// TIA Portal project "May dong chai_PLC_TiaPortal" (V16)
// Vorlageprojekt für das Buch mit Zielsystem S7-1200

(* hardware
DEVICE "S7-1200-Station_1"  S7-1200 Station
   slot 0: "Baugruppenträger_0"  Rack  V1.0
   slot 1: "PLC_1"  CPU 1211C DC/DC/DC  6ES7 211-1AE40-0XB0  V4.1
*)

// ===== PLC "PLC_1"  CPU 1211C DC/DC/DC =====

VAR_GLOBAL   // PLC tag table "Standard-Variablentabelle"
   "box-conveyor" AT %A0.0 : Bool;
   "start" AT %E0.0 : Bool;
   "stop" AT %E0.1 : Bool;
   "latch-relay" AT %M1.5 : Bool;
   "running" AT %M1.4 : Bool;
   "box-sensor" AT %I0.2 : Bool;
   "stop-state" AT %M1.6 : Bool;
   "can-conveyor" AT %Q0.1 : Bool;
   "can-sensor" AT %I0.3 : Bool;
   "Tag_10" AT %M2.0 : Bool;
   "1s" AT %M0.5 : Bool;
   "stop-light" AT %Q0.2 : Bool;
   "Clock_Byte" AT %MB0 : Byte;
   "Clock_10Hz" AT %M0.0 : Bool;
   "Clock_5Hz" AT %M0.1 : Bool;
   "Clock_2.5Hz" AT %M0.2 : Bool;
   "Clock_2Hz" AT %M0.3 : Bool;
   "Clock_1.25Hz" AT %M0.4 : Bool;
   "Clock_1Hz" AT %M0.5 : Bool;
   "Clock_0.625Hz" AT %M0.6 : Bool;
   "Clock_0.5Hz" AT %M0.7 : Bool;
END_VAR

// folder: System blocks/Program resources

DATA_BLOCK "counter1"   // DB1
{ S7_Optimized_Access := 'TRUE' }
AUTHOR : Simatic
FAMILY : IEC
NAME : CNTR
VERSION : 1.0
// stored: InstanceOfName IEC_COUNTER
"IEC_COUNTER"
BEGIN
END_DATA_BLOCK

DATA_BLOCK "counter2"   // DB2
{ S7_Optimized_Access := 'TRUE' }
AUTHOR : Simatic
FAMILY : IEC
NAME : CNTR
VERSION : 1.0
// stored: InstanceOfName IEC_COUNTER
"IEC_COUNTER"
BEGIN
END_DATA_BLOCK

DATA_BLOCK "timer1"   // DB3
{ S7_Optimized_Access := 'TRUE' }
AUTHOR : Simatic
FAMILY : IEC
NAME : IEC_TMR
VERSION : 1.0
// stored: InstanceOfName IEC_TIMER
"IEC_TIMER"
BEGIN
END_DATA_BLOCK

// folder: (top level)

FUNCTION "MHJ-PLC-Lab-Function-S71200" : Void   // FC9000, SCL
{ S7_Optimized_Access := 'TRUE' }
VERSION : 0.1
   VAR_TEMP
      rdTimeReturn : Int;
      outputTime : DTL;
      SyncVal : Byte;
      forVal : Int;
      forVal_2 : Int;
      Value : Byte;
   END_VAR
   VAR CONSTANT
      CompVal : Byte := 16#34;
      Value_01 : Byte := 16#11;
      Value_01_DW : DWord := 16#A165_D992;
      Value_02_DW : DWord := 16#58BE_4401;
   END_VAR
BEGIN

   #Value:=PEEK(area := 16#82,
        dbNumber := 0,
        byteOffset := 511);
   #Value := #Value + 1;

   POKE(area := 16#82,
        dbNumber := 0,
        byteOffset := 511,
        value := #Value);

   POKE(area:=16#81,
        dbNumber:=0,
        byteOffset:=1016,
        value:=#Value_01_DW);
   POKE(area := 16#81,
        dbNumber := 0,
        byteOffset := 1020,
        value := #Value_02_DW);

   POKE(area := 16#81,
        dbNumber := 0,
        byteOffset := 511,
        value := B#16#00);

   FOR #forVal := 0 TO 120 DO
       FOR #forVal_2:=0 TO 10 DO
           #rdTimeReturn:=RD_SYS_T(#outputTime);
           #rdTimeReturn := WR_SYS_T(#outputTime);
           #rdTimeReturn := RD_SYS_T(#outputTime);
           #rdTimeReturn := WR_SYS_T(#outputTime);
       END_FOR;
       #SyncVal:= PEEK(area := 16#81,
                      dbNumber := 0,
                      byteOffset := 511);
       IF #SyncVal = #CompVal THEN
          GOTO M_1;
       END_IF;
   END_FOR;
   RETURN;

   M_1:
   POKE(area := 16#81,
        dbNumber := 0,
        byteOffset := 511,
        value := B#16#0);
END_FUNCTION

ORGANIZATION_BLOCK "Main"   // OB1, LAD, ProgramCycle
TITLE = "Main Program Sweep (Cycle)"
{ S7_Optimized_Access := 'TRUE' }
VERSION : 0.1
   VAR_INPUT
      Initial_Call : Bool;   // Initial call of this OB
      Remanence : Bool;   // =True, if remanent data are available
   END_VAR
   VAR_TEMP   // added for the SCL form of the ladder/FBD networks
      _w1 : Bool;
      _w2 : Bool;
   END_VAR
BEGIN

REGION Network 1: Konnektierungsbaustein für PLC-Lab
   // Im Netzwerk 1 wird der Konnektierungsbaustein für PLC-Lab aufgerufen.
   // Dieser Aufruf darf nicht entfernt werden!
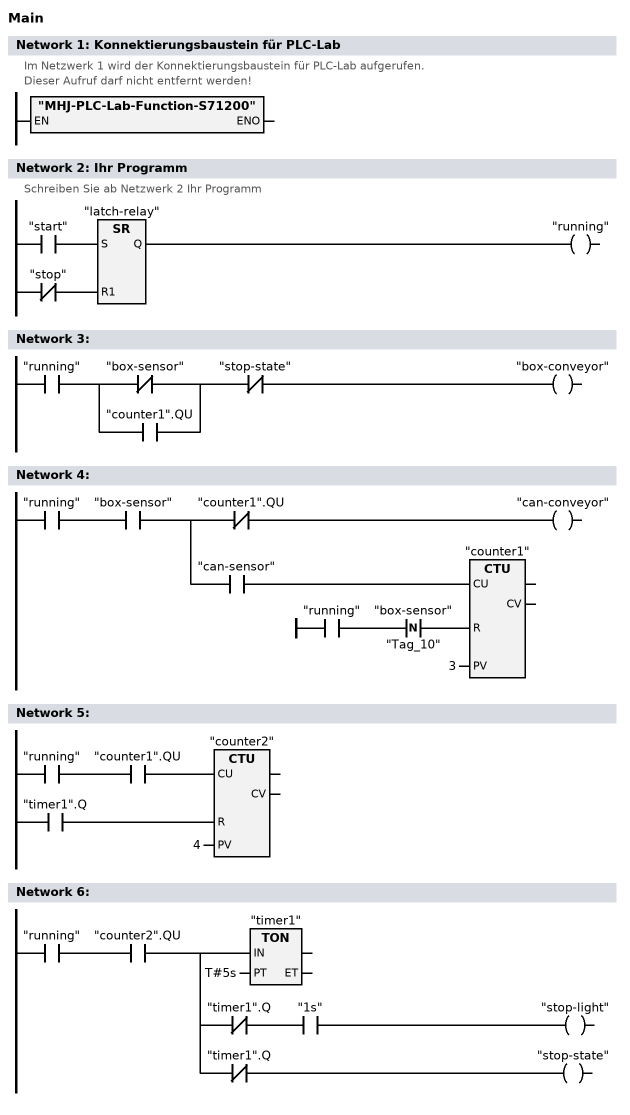
   RUNG wire#powerrail
      "MHJ-PLC-Lab-Function-S71200"()
   END_RUNG
   // the same network as SCL:
   "MHJ-PLC-Lab-Function-S71200"();
END_REGION

REGION Network 2: Ihr Programm
   // Schreiben Sie ab Netzwerk 2 Ihr Programm
   RUNG wire#powerrail
      Contact( "start" )
      S_SR(operand := "latch-relay", r1 := wire#w1)
      Coil( "running" )
   END_RUNG
   RUNG wire#powerrail
      I_Contact( "stop" )
   END_RUNG wire#w1
   // the same network as SCL:
   IF "start" THEN
       "latch-relay" := TRUE;   // SR flip-flop
   END_IF;
   IF NOT "stop" THEN "latch-relay" := FALSE; END_IF;
   "running" := "latch-relay";
END_REGION

REGION Network 3
   RUNG wire#powerrail
      Contact( "running" )
      wire#w1
      I_Contact( "box-sensor" )
      wire#w2
      I_Contact( "stop-state" )
      Coil( "box-conveyor" )
   END_RUNG
   RUNG wire#w1
      Contact( "counter1".QU )
   END_RUNG wire#w2
   // the same network as SCL:
   "box-conveyor" := "running" AND (NOT "box-sensor" OR "counter1".QU) AND NOT "stop-state";
END_REGION

REGION Network 4
   #_w1 := "running" AND "box-sensor";
   "can-conveyor" := #_w1 AND NOT "counter1".QU;
   #_w2 := "running" AND NOT "box-sensor" AND "Tag_10";   // falling edge of "box-sensor"
   "Tag_10" := "box-sensor";
   "counter1".CTU(CU := #_w1 AND "can-sensor", R := #_w2, PV := 3);
END_REGION

REGION Network 5
   "counter2".CTU(CU := "running" AND "counter1".QU, R := "timer1".Q, PV := 4);
END_REGION

REGION Network 6
   #_w1 := "running" AND "counter2".QU;
   "timer1".TON(IN := #_w1, PT := T#5s);
   "stop-light" := #_w1 AND NOT "timer1".Q AND "1s";
   "stop-state" := #_w1 AND NOT "timer1".Q;
END_REGION
END_ORGANIZATION_BLOCK